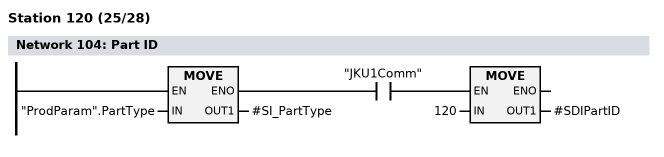
   RUNG wire#powerrail
      Move(in := "ProdParam".PartType, out1 => #SI_PartType)
      Contact( "JKU1Comm" )
      Move(in := 120, out1 => #SDIPartID)
   END_RUNG
   // the same network as SCL:
   #SI_PartType := "ProdParam".PartType;
   IF "JKU1Comm" THEN #SDIPartID := 120; END_IF;
END_REGION

REGION Network 105: Clear positions and map - commands
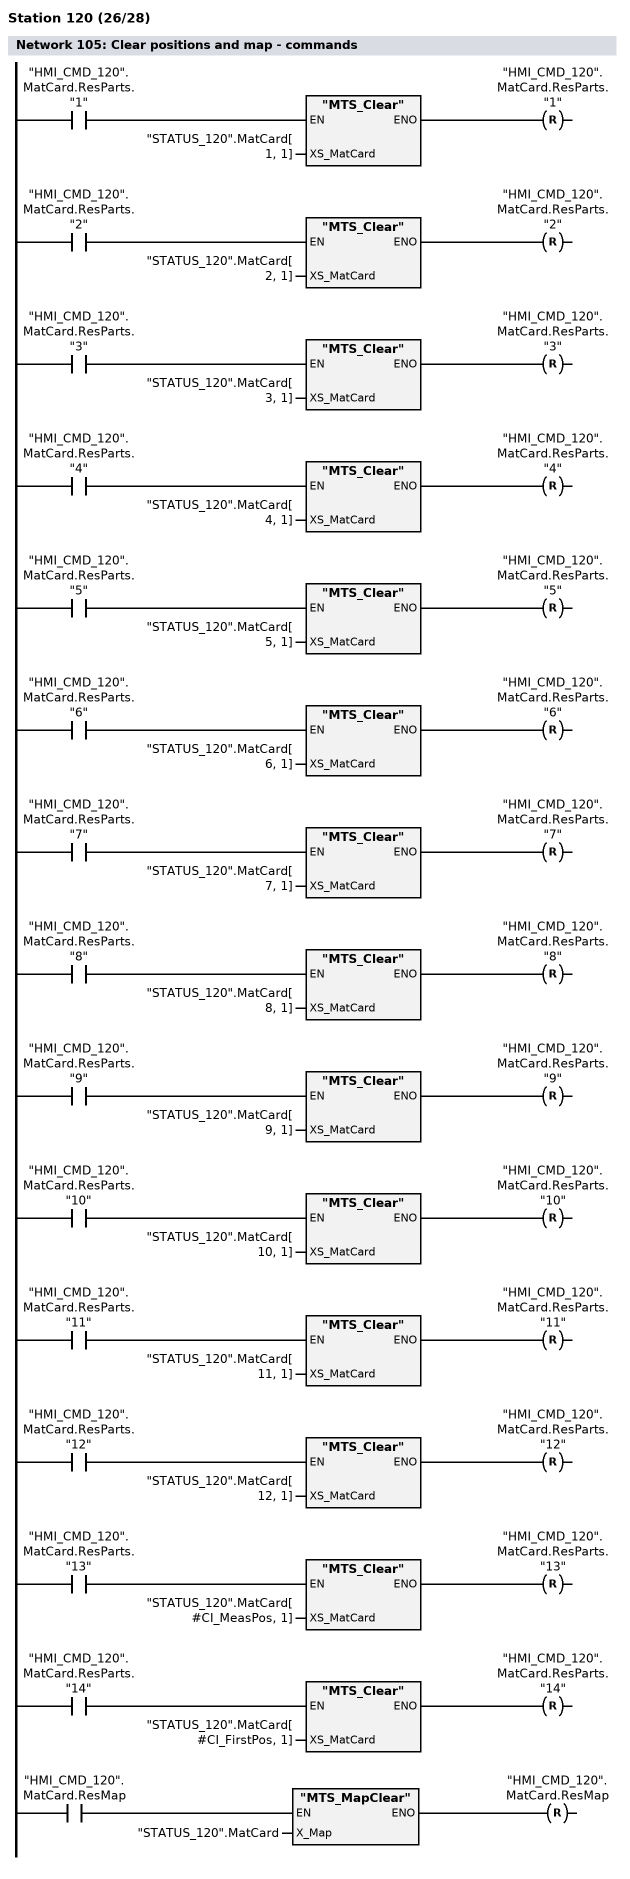
   RUNG wire#powerrail
      Contact( "HMI_CMD_120".MatCard.ResParts."1" )
      "MTS_Clear"(XS_MatCard := "STATUS_120".MatCard[1, 1])
      R_Coil( "HMI_CMD_120".MatCard.ResParts."1" )
   END_RUNG
   RUNG wire#powerrail
      Contact( "HMI_CMD_120".MatCard.ResParts."2" )
      "MTS_Clear"(XS_MatCard := "STATUS_120".MatCard[2, 1])
      R_Coil( "HMI_CMD_120".MatCard.ResParts."2" )
   END_RUNG
   RUNG wire#powerrail
      Contact( "HMI_CMD_120".MatCard.ResParts."3" )
      "MTS_Clear"(XS_MatCard := "STATUS_120".MatCard[3, 1])
      R_Coil( "HMI_CMD_120".MatCard.ResParts."3" )
   END_RUNG
   RUNG wire#powerrail
      Contact( "HMI_CMD_120".MatCard.ResParts."4" )
      "MTS_Clear"(XS_MatCard := "STATUS_120".MatCard[4, 1])
      R_Coil( "HMI_CMD_120".MatCard.ResParts."4" )
   END_RUNG
   RUNG wire#powerrail
      Contact( "HMI_CMD_120".MatCard.ResParts."5" )
      "MTS_Clear"(XS_MatCard := "STATUS_120".MatCard[5, 1])
      R_Coil( "HMI_CMD_120".MatCard.ResParts."5" )
   END_RUNG
   RUNG wire#powerrail
      Contact( "HMI_CMD_120".MatCard.ResParts."6" )
      "MTS_Clear"(XS_MatCard := "STATUS_120".MatCard[6, 1])
      R_Coil( "HMI_CMD_120".MatCard.ResParts."6" )
   END_RUNG
   RUNG wire#powerrail
      Contact( "HMI_CMD_120".MatCard.ResParts."7" )
      "MTS_Clear"(XS_MatCard := "STATUS_120".MatCard[7, 1])
      R_Coil( "HMI_CMD_120".MatCard.ResParts."7" )
   END_RUNG
   RUNG wire#powerrail
      Contact( "HMI_CMD_120".MatCard.ResParts."8" )
      "MTS_Clear"(XS_MatCard := "STATUS_120".MatCard[8, 1])
      R_Coil( "HMI_CMD_120".MatCard.ResParts."8" )
   END_RUNG
   RUNG wire#powerrail
      Contact( "HMI_CMD_120".MatCard.ResParts."9" )
      "MTS_Clear"(XS_MatCard := "STATUS_120".MatCard[9, 1])
      R_Coil( "HMI_CMD_120".MatCard.ResParts."9" )
   END_RUNG
   RUNG wire#powerrail
      Contact( "HMI_CMD_120".MatCard.ResParts."10" )
      "MTS_Clear"(XS_MatCard := "STATUS_120".MatCard[10, 1])
      R_Coil( "HMI_CMD_120".MatCard.ResParts."10" )
   END_RUNG
   RUNG wire#powerrail
      Contact( "HMI_CMD_120".MatCard.ResParts."11" )
      "MTS_Clear"(XS_MatCard := "STATUS_120".MatCard[11, 1])
      R_Coil( "HMI_CMD_120".MatCard.ResParts."11" )
   END_RUNG
   RUNG wire#powerrail
      Contact( "HMI_CMD_120".MatCard.ResParts."12" )
      "MTS_Clear"(XS_MatCard := "STATUS_120".MatCard[12, 1])
      R_Coil( "HMI_CMD_120".MatCard.ResParts."12" )
   END_RUNG
   RUNG wire#powerrail
      Contact( "HMI_CMD_120".MatCard.ResParts."13" )
      "MTS_Clear"(XS_MatCard := "STATUS_120".MatCard[#CI_MeasPos, 1])
      R_Coil( "HMI_CMD_120".MatCard.ResParts."13" )
   END_RUNG
   RUNG wire#powerrail
      Contact( "HMI_CMD_120".MatCard.ResParts."14" )
      "MTS_Clear"(XS_MatCard := "STATUS_120".MatCard[#CI_FirstPos, 1])
      R_Coil( "HMI_CMD_120".MatCard.ResParts."14" )
   END_RUNG
   RUNG wire#powerrail
      Contact( "HMI_CMD_120".MatCard.ResMap )
      "MTS_MapClear"(X_Map := "STATUS_120".MatCard)
      R_Coil( "HMI_CMD_120".MatCard.ResMap )
   END_RUNG
   // the same network as SCL:
   "MTS_Clear"(EN := "HMI_CMD_120".MatCard.ResParts."1", XS_MatCard := "STATUS_120".MatCard[1, 1], ENO => #_w1);
   IF #_w1 THEN "HMI_CMD_120".MatCard.ResParts."1" := FALSE; END_IF;
   "MTS_Clear"(EN := "HMI_CMD_120".MatCard.ResParts."2", XS_MatCard := "STATUS_120".MatCard[2, 1], ENO => #_w2);
   IF #_w2 THEN "HMI_CMD_120".MatCard.ResParts."2" := FALSE; END_IF;
   "MTS_Clear"(EN := "HMI_CMD_120".MatCard.ResParts."3", XS_MatCard := "STATUS_120".MatCard[3, 1], ENO => #_w3);
   IF #_w3 THEN "HMI_CMD_120".MatCard.ResParts."3" := FALSE; END_IF;
   "MTS_Clear"(EN := "HMI_CMD_120".MatCard.ResParts."4", XS_MatCard := "STATUS_120".MatCard[4, 1], ENO => #_w4);
   IF #_w4 THEN "HMI_CMD_120".MatCard.ResParts."4" := FALSE; END_IF;
   "MTS_Clear"(EN := "HMI_CMD_120".MatCard.ResParts."5", XS_MatCard := "STATUS_120".MatCard[5, 1], ENO => #_w5);
   IF #_w5 THEN "HMI_CMD_120".MatCard.ResParts."5" := FALSE; END_IF;
   "MTS_Clear"(EN := "HMI_CMD_120".MatCard.ResParts."6", XS_MatCard := "STATUS_120".MatCard[6, 1], ENO => #_w6);
   IF #_w6 THEN "HMI_CMD_120".MatCard.ResParts."6" := FALSE; END_IF;
   "MTS_Clear"(EN := "HMI_CMD_120".MatCard.ResParts."7", XS_MatCard := "STATUS_120".MatCard[7, 1], ENO => #_w7);
   IF #_w7 THEN "HMI_CMD_120".MatCard.ResParts."7" := FALSE; END_IF;
   "MTS_Clear"(EN := "HMI_CMD_120".MatCard.ResParts."8", XS_MatCard := "STATUS_120".MatCard[8, 1], ENO => #_w8);
   IF #_w8 THEN "HMI_CMD_120".MatCard.ResParts."8" := FALSE; END_IF;
   "MTS_Clear"(EN := "HMI_CMD_120".MatCard.ResParts."9", XS_MatCard := "STATUS_120".MatCard[9, 1], ENO => #_w9);
   IF #_w9 THEN "HMI_CMD_120".MatCard.ResParts."9" := FALSE; END_IF;
   "MTS_Clear"(EN := "HMI_CMD_120".MatCard.ResParts."10",
               XS_MatCard := "STATUS_120".MatCard[10, 1],
               ENO => #_w10);
   IF #_w10 THEN "HMI_CMD_120".MatCard.ResParts."10" := FALSE; END_IF;
   "MTS_Clear"(EN := "HMI_CMD_120".MatCard.ResParts."11",
               XS_MatCard := "STATUS_120".MatCard[11, 1],
               ENO => #_w11);
   IF #_w11 THEN "HMI_CMD_120".MatCard.ResParts."11" := FALSE; END_IF;
   "MTS_Clear"(EN := "HMI_CMD_120".MatCard.ResParts."12",
               XS_MatCard := "STATUS_120".MatCard[12, 1],
               ENO => #_w12);
   IF #_w12 THEN "HMI_CMD_120".MatCard.ResParts."12" := FALSE; END_IF;
   "MTS_Clear"(EN := "HMI_CMD_120".MatCard.ResParts."13",
               XS_MatCard := "STATUS_120".MatCard[#CI_MeasPos, 1],
               ENO => #_w13);
   IF #_w13 THEN "HMI_CMD_120".MatCard.ResParts."13" := FALSE; END_IF;
   "MTS_Clear"(EN := "HMI_CMD_120".MatCard.ResParts."14",
               XS_MatCard := "STATUS_120".MatCard[#CI_FirstPos, 1],
               ENO => #_w14);
   IF #_w14 THEN "HMI_CMD_120".MatCard.ResParts."14" := FALSE; END_IF;
   "MTS_MapClear"(EN := "HMI_CMD_120".MatCard.ResMap, X_Map := "STATUS_120".MatCard, ENO => #_w15);
   IF #_w15 THEN "HMI_CMD_120".MatCard.ResMap := FALSE; END_IF;
END_REGION

REGION Network 106: Set positions and map - commands
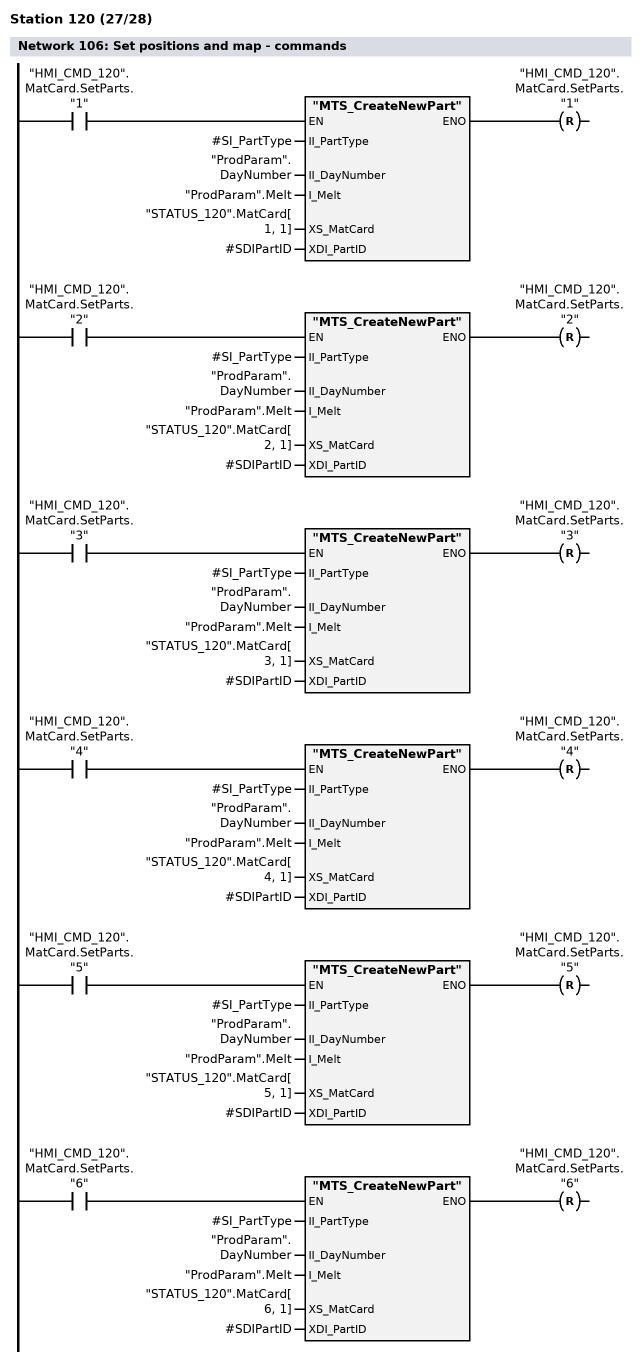
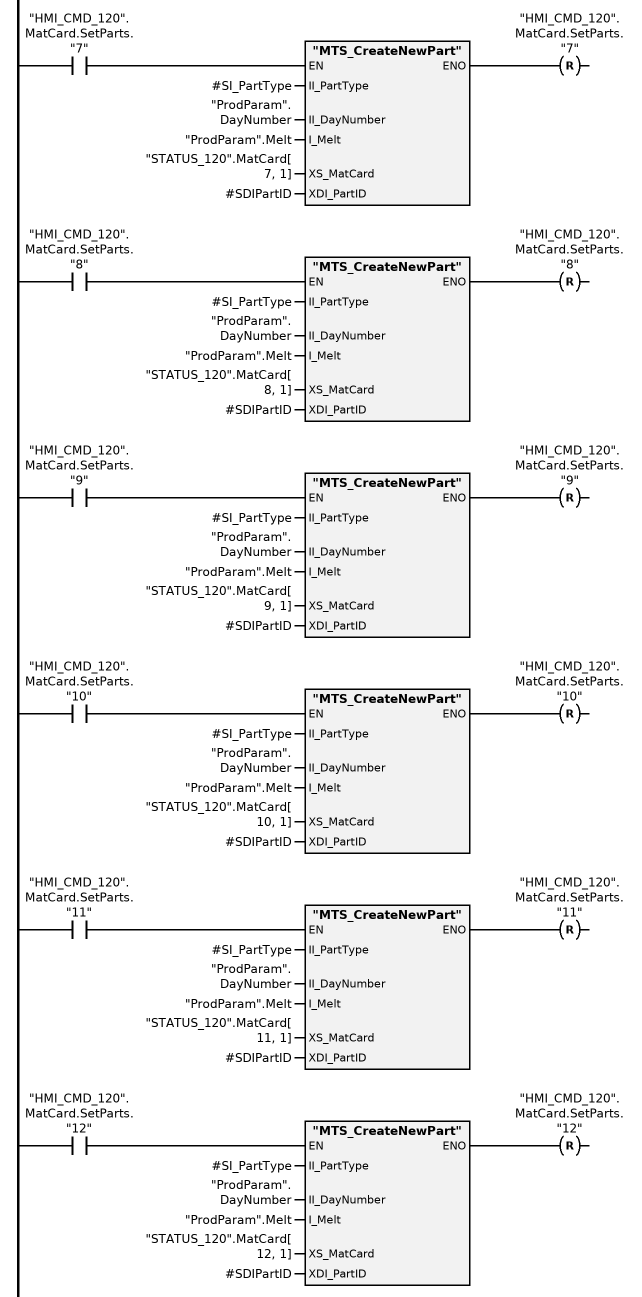
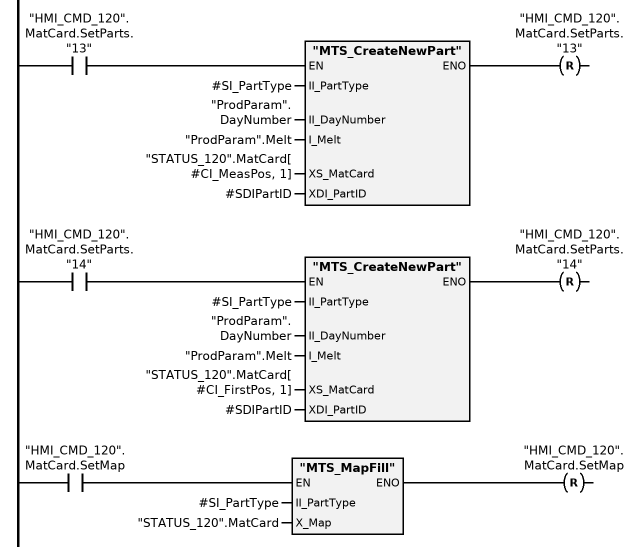
   RUNG wire#powerrail
      Contact( "HMI_CMD_120".MatCard.SetParts."1" )
      "MTS_CreateNewPart"(II_PartType := #SI_PartType, II_DayNumber := "ProdParam".DayNumber, I_Melt := "ProdParam".Melt, XS_MatCard := "STATUS_120".MatCard[1, 1], XDI_PartID := #SDIPartID)
      R_Coil( "HMI_CMD_120".MatCard.SetParts."1" )
   END_RUNG
   RUNG wire#powerrail
      Contact( "HMI_CMD_120".MatCard.SetParts."2" )
      "MTS_CreateNewPart"(II_PartType := #SI_PartType, II_DayNumber := "ProdParam".DayNumber, I_Melt := "ProdParam".Melt, XS_MatCard := "STATUS_120".MatCard[2, 1], XDI_PartID := #SDIPartID)
      R_Coil( "HMI_CMD_120".MatCard.SetParts."2" )
   END_RUNG
   RUNG wire#powerrail
      Contact( "HMI_CMD_120".MatCard.SetParts."3" )
      "MTS_CreateNewPart"(II_PartType := #SI_PartType, II_DayNumber := "ProdParam".DayNumber, I_Melt := "ProdParam".Melt, XS_MatCard := "STATUS_120".MatCard[3, 1], XDI_PartID := #SDIPartID)
      R_Coil( "HMI_CMD_120".MatCard.SetParts."3" )
   END_RUNG
   RUNG wire#powerrail
      Contact( "HMI_CMD_120".MatCard.SetParts."4" )
      "MTS_CreateNewPart"(II_PartType := #SI_PartType, II_DayNumber := "ProdParam".DayNumber, I_Melt := "ProdParam".Melt, XS_MatCard := "STATUS_120".MatCard[4, 1], XDI_PartID := #SDIPartID)
      R_Coil( "HMI_CMD_120".MatCard.SetParts."4" )
   END_RUNG
   RUNG wire#powerrail
      Contact( "HMI_CMD_120".MatCard.SetParts."5" )
      "MTS_CreateNewPart"(II_PartType := #SI_PartType, II_DayNumber := "ProdParam".DayNumber, I_Melt := "ProdParam".Melt, XS_MatCard := "STATUS_120".MatCard[5, 1], XDI_PartID := #SDIPartID)
      R_Coil( "HMI_CMD_120".MatCard.SetParts."5" )
   END_RUNG
   RUNG wire#powerrail
      Contact( "HMI_CMD_120".MatCard.SetParts."6" )
      "MTS_CreateNewPart"(II_PartType := #SI_PartType, II_DayNumber := "ProdParam".DayNumber, I_Melt := "ProdParam".Melt, XS_MatCard := "STATUS_120".MatCard[6, 1], XDI_PartID := #SDIPartID)
      R_Coil( "HMI_CMD_120".MatCard.SetParts."6" )
   END_RUNG
   RUNG wire#powerrail
      Contact( "HMI_CMD_120".MatCard.SetParts."7" )
      "MTS_CreateNewPart"(II_PartType := #SI_PartType, II_DayNumber := "ProdParam".DayNumber, I_Melt := "ProdParam".Melt, XS_MatCard := "STATUS_120".MatCard[7, 1], XDI_PartID := #SDIPartID)
      R_Coil( "HMI_CMD_120".MatCard.SetParts."7" )
   END_RUNG
   RUNG wire#powerrail
      Contact( "HMI_CMD_120".MatCard.SetParts."8" )
      "MTS_CreateNewPart"(II_PartType := #SI_PartType, II_DayNumber := "ProdParam".DayNumber, I_Melt := "ProdParam".Melt, XS_MatCard := "STATUS_120".MatCard[8, 1], XDI_PartID := #SDIPartID)
      R_Coil( "HMI_CMD_120".MatCard.SetParts."8" )
   END_RUNG
   RUNG wire#powerrail
      Contact( "HMI_CMD_120".MatCard.SetParts."9" )
      "MTS_CreateNewPart"(II_PartType := #SI_PartType, II_DayNumber := "ProdParam".DayNumber, I_Melt := "ProdParam".Melt, XS_MatCard := "STATUS_120".MatCard[9, 1], XDI_PartID := #SDIPartID)
      R_Coil( "HMI_CMD_120".MatCard.SetParts."9" )
   END_RUNG
   RUNG wire#powerrail
      Contact( "HMI_CMD_120".MatCard.SetParts."10" )
      "MTS_CreateNewPart"(II_PartType := #SI_PartType, II_DayNumber := "ProdParam".DayNumber, I_Melt := "ProdParam".Melt, XS_MatCard := "STATUS_120".MatCard[10, 1], XDI_PartID := #SDIPartID)
      R_Coil( "HMI_CMD_120".MatCard.SetParts."10" )
   END_RUNG
   RUNG wire#powerrail
      Contact( "HMI_CMD_120".MatCard.SetParts."11" )
      "MTS_CreateNewPart"(II_PartType := #SI_PartType, II_DayNumber := "ProdParam".DayNumber, I_Melt := "ProdParam".Melt, XS_MatCard := "STATUS_120".MatCard[11, 1], XDI_PartID := #SDIPartID)
      R_Coil( "HMI_CMD_120".MatCard.SetParts."11" )
   END_RUNG
   RUNG wire#powerrail
      Contact( "HMI_CMD_120".MatCard.SetParts."12" )
      "MTS_CreateNewPart"(II_PartType := #SI_PartType, II_DayNumber := "ProdParam".DayNumber, I_Melt := "ProdParam".Melt, XS_MatCard := "STATUS_120".MatCard[12, 1], XDI_PartID := #SDIPartID)
      R_Coil( "HMI_CMD_120".MatCard.SetParts."12" )
   END_RUNG
   RUNG wire#powerrail
      Contact( "HMI_CMD_120".MatCard.SetParts."13" )
      "MTS_CreateNewPart"(II_PartType := #SI_PartType, II_DayNumber := "ProdParam".DayNumber, I_Melt := "ProdParam".Melt, XS_MatCard := "STATUS_120".MatCard[#CI_MeasPos, 1], XDI_PartID := #SDIPartID)
      R_Coil( "HMI_CMD_120".MatCard.SetParts."13" )
   END_RUNG
   RUNG wire#powerrail
      Contact( "HMI_CMD_120".MatCard.SetParts."14" )
      "MTS_CreateNewPart"(II_PartType := #SI_PartType, II_DayNumber := "ProdParam".DayNumber, I_Melt := "ProdParam".Melt, XS_MatCard := "STATUS_120".MatCard[#CI_FirstPos, 1], XDI_PartID := #SDIPartID)
      R_Coil( "HMI_CMD_120".MatCard.SetParts."14" )
   END_RUNG
   RUNG wire#powerrail
      Contact( "HMI_CMD_120".MatCard.SetMap )
      "MTS_MapFill"(II_PartType := #SI_PartType, X_Map := "STATUS_120".MatCard)
      R_Coil( "HMI_CMD_120".MatCard.SetMap )
   END_RUNG
   // the same network as SCL:
   "MTS_CreateNewPart"(EN := "HMI_CMD_120".MatCard.SetParts."1",
                       II_PartType := #SI_PartType,
                       II_DayNumber := "ProdParam".DayNumber,
                       I_Melt := "ProdParam".Melt,
                       XS_MatCard := "STATUS_120".MatCard[1, 1],
                       XDI_PartID := #SDIPartID,
                       ENO => #_w1);
   IF #_w1 THEN "HMI_CMD_120".MatCard.SetParts."1" := FALSE; END_IF;
   "MTS_CreateNewPart"(EN := "HMI_CMD_120".MatCard.SetParts."2",
                       II_PartType := #SI_PartType,
                       II_DayNumber := "ProdParam".DayNumber,
                       I_Melt := "ProdParam".Melt,
                       XS_MatCard := "STATUS_120".MatCard[2, 1],
                       XDI_PartID := #SDIPartID,
                       ENO => #_w2);
   IF #_w2 THEN "HMI_CMD_120".MatCard.SetParts."2" := FALSE; END_IF;
   "MTS_CreateNewPart"(EN := "HMI_CMD_120".MatCard.SetParts."3",
                       II_PartType := #SI_PartType,
                       II_DayNumber := "ProdParam".DayNumber,
                       I_Melt := "ProdParam".Melt,
                       XS_MatCard := "STATUS_120".MatCard[3, 1],
                       XDI_PartID := #SDIPartID,
                       ENO => #_w3);
   IF #_w3 THEN "HMI_CMD_120".MatCard.SetParts."3" := FALSE; END_IF;
   "MTS_CreateNewPart"(EN := "HMI_CMD_120".MatCard.SetParts."4",
                       II_PartType := #SI_PartType,
                       II_DayNumber := "ProdParam".DayNumber,
                       I_Melt := "ProdParam".Melt,
                       XS_MatCard := "STATUS_120".MatCard[4, 1],
                       XDI_PartID := #SDIPartID,
                       ENO => #_w4);
   IF #_w4 THEN "HMI_CMD_120".MatCard.SetParts."4" := FALSE; END_IF;
   "MTS_CreateNewPart"(EN := "HMI_CMD_120".MatCard.SetParts."5",
                       II_PartType := #SI_PartType,
                       II_DayNumber := "ProdParam".DayNumber,
                       I_Melt := "ProdParam".Melt,
                       XS_MatCard := "STATUS_120".MatCard[5, 1],
                       XDI_PartID := #SDIPartID,
                       ENO => #_w5);
   IF #_w5 THEN "HMI_CMD_120".MatCard.SetParts."5" := FALSE; END_IF;
   "MTS_CreateNewPart"(EN := "HMI_CMD_120".MatCard.SetParts."6",
                       II_PartType := #SI_PartType,
                       II_DayNumber := "ProdParam".DayNumber,
                       I_Melt := "ProdParam".Melt,
                       XS_MatCard := "STATUS_120".MatCard[6, 1],
                       XDI_PartID := #SDIPartID,
                       ENO => #_w6);
   IF #_w6 THEN "HMI_CMD_120".MatCard.SetParts."6" := FALSE; END_IF;
   "MTS_CreateNewPart"(EN := "HMI_CMD_120".MatCard.SetParts."7",
                       II_PartType := #SI_PartType,
                       II_DayNumber := "ProdParam".DayNumber,
                       I_Melt := "ProdParam".Melt,
                       XS_MatCard := "STATUS_120".MatCard[7, 1],
                       XDI_PartID := #SDIPartID,
                       ENO => #_w7);
   IF #_w7 THEN "HMI_CMD_120".MatCard.SetParts."7" := FALSE; END_IF;
   "MTS_CreateNewPart"(EN := "HMI_CMD_120".MatCard.SetParts."8",
                       II_PartType := #SI_PartType,
                       II_DayNumber := "ProdParam".DayNumber,
                       I_Melt := "ProdParam".Melt,
                       XS_MatCard := "STATUS_120".MatCard[8, 1],
                       XDI_PartID := #SDIPartID,
                       ENO => #_w8);
   IF #_w8 THEN "HMI_CMD_120".MatCard.SetParts."8" := FALSE; END_IF;
   "MTS_CreateNewPart"(EN := "HMI_CMD_120".MatCard.SetParts."9",
                       II_PartType := #SI_PartType,
                       II_DayNumber := "ProdParam".DayNumber,
                       I_Melt := "ProdParam".Melt,
                       XS_MatCard := "STATUS_120".MatCard[9, 1],
                       XDI_PartID := #SDIPartID,
                       ENO => #_w9);
   IF #_w9 THEN "HMI_CMD_120".MatCard.SetParts."9" := FALSE; END_IF;
   "MTS_CreateNewPart"(EN := "HMI_CMD_120".MatCard.SetParts."10",
                       II_PartType := #SI_PartType,
                       II_DayNumber := "ProdParam".DayNumber,
                       I_Melt := "ProdParam".Melt,
                       XS_MatCard := "STATUS_120".MatCard[10, 1],
                       XDI_PartID := #SDIPartID,
                       ENO => #_w10);
   IF #_w10 THEN "HMI_CMD_120".MatCard.SetParts."10" := FALSE; END_IF;
   "MTS_CreateNewPart"(EN := "HMI_CMD_120".MatCard.SetParts."11",
                       II_PartType := #SI_PartType,
                       II_DayNumber := "ProdParam".DayNumber,
                       I_Melt := "ProdParam".Melt,
                       XS_MatCard := "STATUS_120".MatCard[11, 1],
                       XDI_PartID := #SDIPartID,
                       ENO => #_w11);
   IF #_w11 THEN "HMI_CMD_120".MatCard.SetParts."11" := FALSE; END_IF;
   "MTS_CreateNewPart"(EN := "HMI_CMD_120".MatCard.SetParts."12",
                       II_PartType := #SI_PartType,
                       II_DayNumber := "ProdParam".DayNumber,
                       I_Melt := "ProdParam".Melt,
                       XS_MatCard := "STATUS_120".MatCard[12, 1],
                       XDI_PartID := #SDIPartID,
                       ENO => #_w12);
   IF #_w12 THEN "HMI_CMD_120".MatCard.SetParts."12" := FALSE; END_IF;
   "MTS_CreateNewPart"(EN := "HMI_CMD_120".MatCard.SetParts."13",
                       II_PartType := #SI_PartType,
                       II_DayNumber := "ProdParam".DayNumber,
                       I_Melt := "ProdParam".Melt,
                       XS_MatCard := "STATUS_120".MatCard[#CI_MeasPos, 1],
                       XDI_PartID := #SDIPartID,
                       ENO => #_w13);
   IF #_w13 THEN "HMI_CMD_120".MatCard.SetParts."13" := FALSE; END_IF;
   "MTS_CreateNewPart"(EN := "HMI_CMD_120".MatCard.SetParts."14",
                       II_PartType := #SI_PartType,
                       II_DayNumber := "ProdParam".DayNumber,
                       I_Melt := "ProdParam".Melt,
                       XS_MatCard := "STATUS_120".MatCard[#CI_FirstPos, 1],
                       XDI_PartID := #SDIPartID,
                       ENO => #_w14);
   IF #_w14 THEN "HMI_CMD_120".MatCard.SetParts."14" := FALSE; END_IF;
   "MTS_MapFill"(EN := "HMI_CMD_120".MatCard.SetMap,
                 II_PartType := #SI_PartType,
                 X_Map := "STATUS_120".MatCard,
                 ENO => #_w15);
   IF #_w15 THEN "HMI_CMD_120".MatCard.SetMap := FALSE; END_IF;
END_REGION

REGION Network 107: Data transfer: KAS2 -> 120 (create new part)
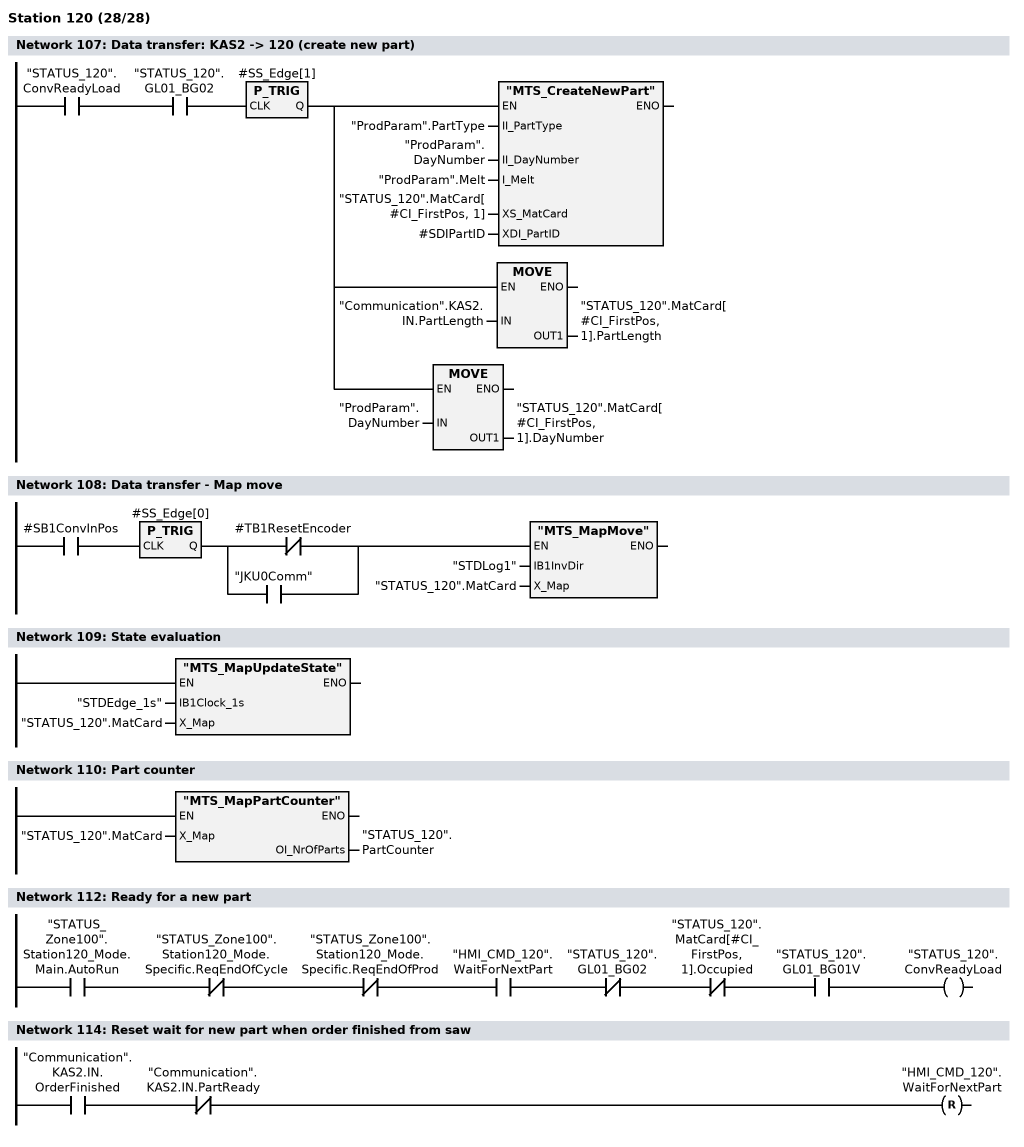
   RUNG wire#powerrail
      Contact( "STATUS_120".ConvReadyLoad )
      Contact( "STATUS_120".GL01_BG02 )
      P_Trig( #SS_Edge[1] )
      wire#w1
      "MTS_CreateNewPart"(II_PartType := "ProdParam".PartType, II_DayNumber := "ProdParam".DayNumber, I_Melt := "ProdParam".Melt, XS_MatCard := "STATUS_120".MatCard[#CI_FirstPos, 1], XDI_PartID := #SDIPartID)
   END_RUNG
   RUNG wire#w1
      Move(in := "Communication".KAS2.IN.PartLength, out1 => "STATUS_120".MatCard[#CI_FirstPos, 1].PartLength)
   END_RUNG
   RUNG wire#w1
      Move(in := "ProdParam".DayNumber, out1 => "STATUS_120".MatCard[#CI_FirstPos, 1].DayNumber)
   END_RUNG
   // the same network as SCL:
   #_w1 := "STATUS_120".ConvReadyLoad AND "STATUS_120".GL01_BG02;
   #_w2 := #_w1 AND NOT #SS_Edge[1];   // rising edge
   #SS_Edge[1] := #_w1;
   IF #_w2 THEN
       "MTS_CreateNewPart"(II_PartType := "ProdParam".PartType,
                           II_DayNumber := "ProdParam".DayNumber,
                           I_Melt := "ProdParam".Melt,
                           XS_MatCard := "STATUS_120".MatCard[#CI_FirstPos, 1],
                           XDI_PartID := #SDIPartID);
       "STATUS_120".MatCard[#CI_FirstPos, 1].PartLength := "Communication".KAS2.IN.PartLength;
       "STATUS_120".MatCard[#CI_FirstPos, 1].DayNumber := "ProdParam".DayNumber;
   END_IF;
END_REGION

REGION Network 108: Data transfer - Map move
   RUNG wire#powerrail
      Contact( #SB1ConvInPos )
      P_Trig( #SS_Edge[0] )
      wire#w1
      I_Contact( #TB1ResetEncoder )
      wire#w2
      "MTS_MapMove"(IB1InvDir := "STDLog1", X_Map := "STATUS_120".MatCard)
   END_RUNG
   RUNG wire#w1
      Contact( "JKU0Comm" )
   END_RUNG wire#w2
   // the same network as SCL:
   #_w1 := #SB1ConvInPos AND NOT #SS_Edge[0];   // rising edge
   #SS_Edge[0] := #SB1ConvInPos;
   IF #_w1 AND (NOT #TB1ResetEncoder OR "JKU0Comm") THEN
       "MTS_MapMove"(IB1InvDir := "STDLog1", X_Map := "STATUS_120".MatCard);
   END_IF;
END_REGION

REGION Network 109: State evaluation
   RUNG wire#powerrail
      "MTS_MapUpdateState"(IB1Clock_1s := "STDEdge_1s", X_Map := "STATUS_120".MatCard)
   END_RUNG
   // the same network as SCL:
   "MTS_MapUpdateState"(IB1Clock_1s := "STDEdge_1s", X_Map := "STATUS_120".MatCard);
END_REGION

REGION Network 110: Part counter
   RUNG wire#powerrail
      "MTS_MapPartCounter"(X_Map := "STATUS_120".MatCard, OI_NrOfParts => "STATUS_120".PartCounter)
   END_RUNG
   // the same network as SCL:
   "MTS_MapPartCounter"(X_Map := "STATUS_120".MatCard, OI_NrOfParts => "STATUS_120".PartCounter);
END_REGION

REGION Network 111: *************** Interface to KAS2 ***************
END_REGION

REGION Network 112: Ready for a new part
   RUNG wire#powerrail
      Contact( "STATUS_Zone100".Station120_Mode.Main.AutoRun )
      I_Contact( "STATUS_Zone100".Station120_Mode.Specific.ReqEndOfCycle )
      I_Contact( "STATUS_Zone100".Station120_Mode.Specific.ReqEndOfProd )
      Contact( "HMI_CMD_120".WaitForNextPart )
      I_Contact( "STATUS_120".GL01_BG02 )
      I_Contact( "STATUS_120".MatCard[#CI_FirstPos, 1].Occupied )
      Contact( "STATUS_120".GL01_BG01V )
      Coil( "STATUS_120".ConvReadyLoad )
   END_RUNG
   // the same network as SCL:
   "STATUS_120".ConvReadyLoad := "STATUS_Zone100".Station120_Mode.Main.AutoRun AND NOT "STATUS_Zone100".Station120_Mode.Specific.ReqEndOfCycle AND NOT "STATUS_Zone100".Station120_Mode.Specific.ReqEndOfProd AND "HMI_CMD_120".WaitForNextPart AND NOT "STATUS_120".GL01_BG02 AND NOT "STATUS_120".MatCard[#CI_FirstPos, 1].Occupied AND "STATUS_120".GL01_BG01V;
END_REGION

REGION Network 113: *************** Aux ***************
END_REGION

REGION Network 114: Reset wait for new part when order finished from saw
   RUNG wire#powerrail
      Contact( "Communication".KAS2.IN.OrderFinished )
      I_Contact( "Communication".KAS2.IN.PartReady )
      R_Coil( "HMI_CMD_120".WaitForNextPart )
   END_RUNG
   // the same network as SCL:
   IF "Communication".KAS2.IN.OrderFinished AND NOT "Communication".KAS2.IN.PartReady THEN
       "HMI_CMD_120".WaitForNextPart := FALSE;
   END_IF;
END_REGION
END_FUNCTION_BLOCK
